// TIA Portal V20 export
TYPE "UDT_AxisPosition"
   STRUCT
      Axis_U : Struct
         PosExternalLoadUnload : Real;
         PosExternalLoadUnloadManu : Real;
         PosPartControl : Real;
         PosBwControl : Real;
         PosInternalLoadUnload : Real;
         PosExtGateExt : Real;
         PosIntGateExt : Real;
         PosExtGateInt : Real;
         PosIntGateInt : Real;
      END_STRUCT;
      Axis_V : Struct
         PosLoadUnload : Real;
         PosSafe : Real;
      END_STRUCT;
      Axis_W : Struct
         PosLoadUnload : Real;
         PosSafe : Real;
         PosApproach : Real;
      END_STRUCT;
   END_STRUCT;
END_TYPE
